// TIA Portal V18 export
// export: Created 2026-06-08T13:24:30.7103891Z, ExportSetting WithDefaults, DisplayName Totally Integrated Automation Portal, DisplayVersion V18, DisplayName TIA Portal Openness, DisplayVersion V18, DisplayName TIA Portal Version Control Interface, DisplayVersion V18, DisplayName STEP 7 Professional, DisplayVersion V18, DisplayName STEP 7 Safety, DisplayVersion V18, DisplayName WinCC Professional, DisplayVersion V18
ORGANIZATION_BLOCK "Main"   // OB1, LAD, ProgramCycle
TITLE = "Main Program Sweep (Cycle)"
{ S7_Optimized_Access := 'TRUE' }
VERSION : 0.1
// stored: AutoNumber true, IsIECCheckEnabled false, SetENOAutomatically false
   VAR_INPUT
      Initial_Call : Bool;   // Initial call of this OB
      Remanence : Bool;   // =True, if remanent data are available
   END_VAR
BEGIN

REGION Network 1: Modbus TCP Server - Call MB_SERVER
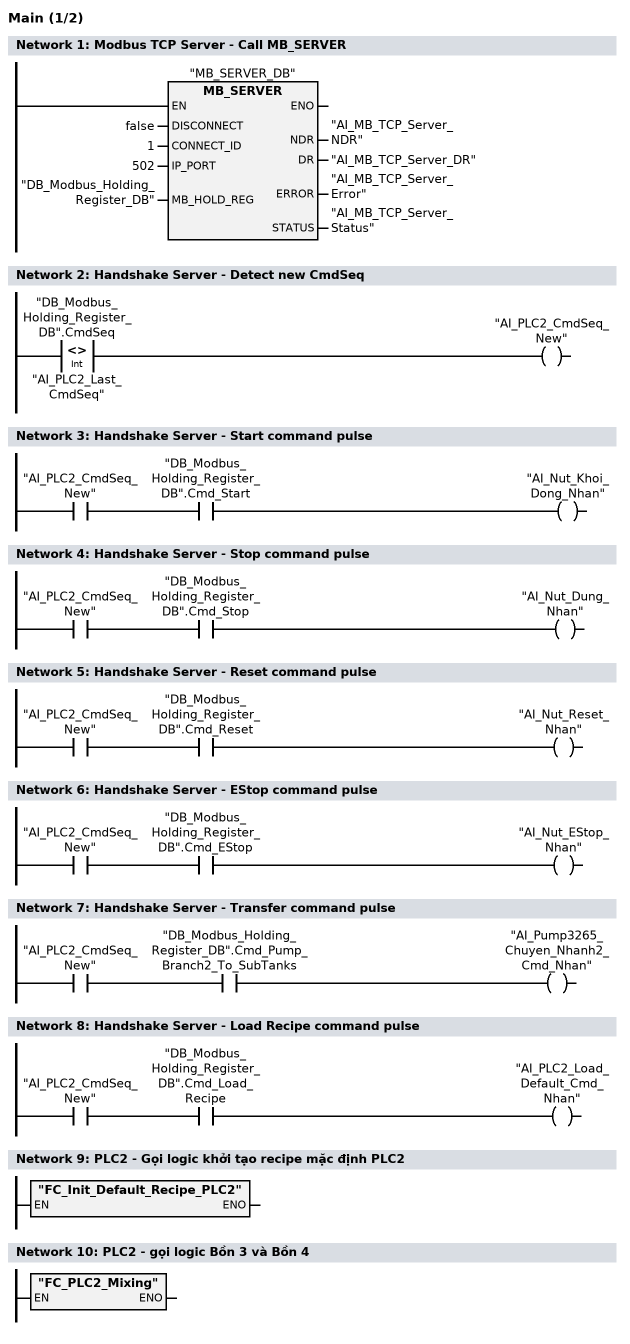
   RUNG wire#powerrail
      { S7_Templates := "[card1200 := 1, card1500 := 0]" } "MB_SERVER_DB".MB_SERVER(DISCONNECT := false, CONNECT_ID := 1, IP_PORT := 502, MB_HOLD_REG := "DB_Modbus_Holding_Register_DB", NDR => "AI_MB_TCP_Server_NDR", DR => "AI_MB_TCP_Server_DR", ERROR => "AI_MB_TCP_Server_Error", STATUS => "AI_MB_TCP_Server_Status")
   END_RUNG
   // the same network as SCL:
   "MB_SERVER_DB"(DISCONNECT := false,   // MB_SERVER
                  CONNECT_ID := 1,
                  IP_PORT := 502,
                  MB_HOLD_REG := "DB_Modbus_Holding_Register_DB",
                  NDR => "AI_MB_TCP_Server_NDR",
                  DR => "AI_MB_TCP_Server_DR",
                  ERROR => "AI_MB_TCP_Server_Error",
                  STATUS => "AI_MB_TCP_Server_Status");
END_REGION

REGION Network 2: Handshake Server - Detect new CmdSeq
   RUNG wire#powerrail
      { S7_Templates := "SrcType := Int" } NE_Contact(in1 := "DB_Modbus_Holding_Register_DB".CmdSeq, in2 := "AI_PLC2_Last_CmdSeq")
      Coil( "AI_PLC2_CmdSeq_New" )
   END_RUNG
   // the same network as SCL:
   "AI_PLC2_CmdSeq_New" := "DB_Modbus_Holding_Register_DB".CmdSeq <> "AI_PLC2_Last_CmdSeq";
END_REGION

REGION Network 3: Handshake Server - Start command pulse
   RUNG wire#powerrail
      Contact( "AI_PLC2_CmdSeq_New" )
      Contact( "DB_Modbus_Holding_Register_DB".Cmd_Start )
      Coil( "AI_Nut_Khoi_Dong_Nhan" )
   END_RUNG
   // the same network as SCL:
   "AI_Nut_Khoi_Dong_Nhan" := "AI_PLC2_CmdSeq_New" AND "DB_Modbus_Holding_Register_DB".Cmd_Start;
END_REGION

REGION Network 4: Handshake Server - Stop command pulse
   RUNG wire#powerrail
      Contact( "AI_PLC2_CmdSeq_New" )
      Contact( "DB_Modbus_Holding_Register_DB".Cmd_Stop )
      Coil( "AI_Nut_Dung_Nhan" )
   END_RUNG
   // the same network as SCL:
   "AI_Nut_Dung_Nhan" := "AI_PLC2_CmdSeq_New" AND "DB_Modbus_Holding_Register_DB".Cmd_Stop;
END_REGION

REGION Network 5: Handshake Server - Reset command pulse
   RUNG wire#powerrail
      Contact( "AI_PLC2_CmdSeq_New" )
      Contact( "DB_Modbus_Holding_Register_DB".Cmd_Reset )
      Coil( "AI_Nut_Reset_Nhan" )
   END_RUNG
   // the same network as SCL:
   "AI_Nut_Reset_Nhan" := "AI_PLC2_CmdSeq_New" AND "DB_Modbus_Holding_Register_DB".Cmd_Reset;
END_REGION

REGION Network 6: Handshake Server - EStop command pulse
   RUNG wire#powerrail
      Contact( "AI_PLC2_CmdSeq_New" )
      Contact( "DB_Modbus_Holding_Register_DB".Cmd_EStop )
      Coil( "AI_Nut_EStop_Nhan" )
   END_RUNG
   // the same network as SCL:
   "AI_Nut_EStop_Nhan" := "AI_PLC2_CmdSeq_New" AND "DB_Modbus_Holding_Register_DB".Cmd_EStop;
END_REGION

REGION Network 7: Handshake Server - Transfer command pulse
   RUNG wire#powerrail
      Contact( "AI_PLC2_CmdSeq_New" )
      Contact( "DB_Modbus_Holding_Register_DB".Cmd_Pump_Branch2_To_SubTanks )
      Coil( "AI_Pump3265_Chuyen_Nhanh2_Cmd_Nhan" )
   END_RUNG
   // the same network as SCL:
   "AI_Pump3265_Chuyen_Nhanh2_Cmd_Nhan" := "AI_PLC2_CmdSeq_New" AND "DB_Modbus_Holding_Register_DB".Cmd_Pump_Branch2_To_SubTanks;
END_REGION

REGION Network 8: Handshake Server - Load Recipe command pulse
   RUNG wire#powerrail
      Contact( "AI_PLC2_CmdSeq_New" )
      Contact( "DB_Modbus_Holding_Register_DB".Cmd_Load_Recipe )
      Coil( "AI_PLC2_Load_Default_Cmd_Nhan" )
   END_RUNG
   // the same network as SCL:
   "AI_PLC2_Load_Default_Cmd_Nhan" := "AI_PLC2_CmdSeq_New" AND "DB_Modbus_Holding_Register_DB".Cmd_Load_Recipe;
END_REGION

REGION Network 9: PLC2 - Gọi logic khởi tạo recipe mặc định PLC2
   RUNG wire#powerrail
      "FC_Init_Default_Recipe_PLC2"()
   END_RUNG
   // the same network as SCL:
   "FC_Init_Default_Recipe_PLC2"();
END_REGION

REGION Network 10: PLC2 - gọi logic Bồn 3 và Bồn 4
   RUNG wire#powerrail
      "FC_PLC2_Mixing"()
   END_RUNG
   // the same network as SCL:
   "FC_PLC2_Mixing"();
END_REGION

REGION Network 11: PLC2 - cập nhật mirror HMI
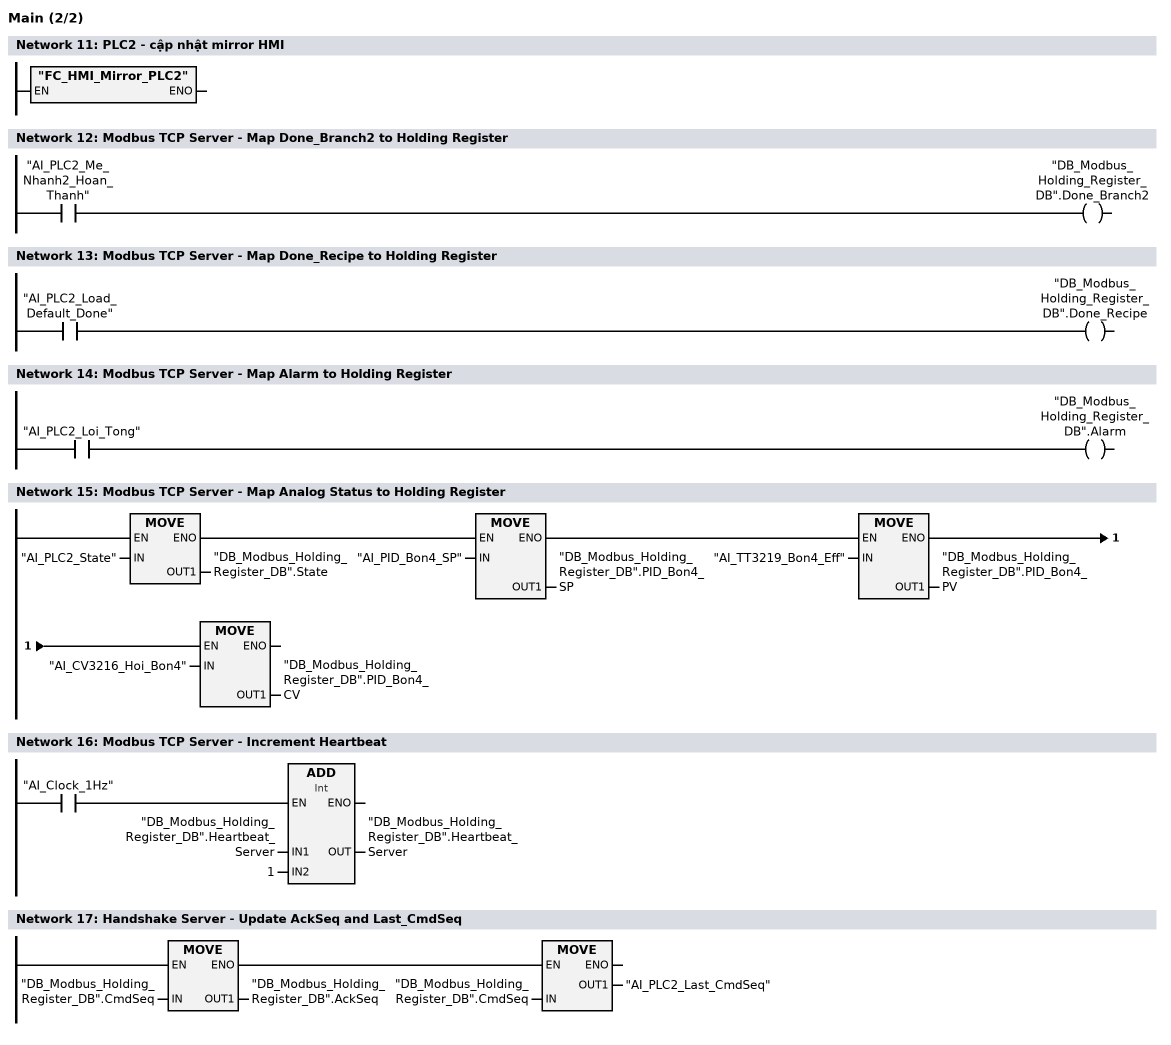
   RUNG wire#powerrail
      "FC_HMI_Mirror_PLC2"()
   END_RUNG
   // the same network as SCL:
   "FC_HMI_Mirror_PLC2"();
END_REGION

REGION Network 12: Modbus TCP Server - Map Done_Branch2 to Holding Register
   RUNG wire#powerrail
      Contact( "AI_PLC2_Me_Nhanh2_Hoan_Thanh" )
      Coil( "DB_Modbus_Holding_Register_DB".Done_Branch2 )
   END_RUNG
   // the same network as SCL:
   "DB_Modbus_Holding_Register_DB".Done_Branch2 := "AI_PLC2_Me_Nhanh2_Hoan_Thanh";
END_REGION

REGION Network 13: Modbus TCP Server - Map Done_Recipe to Holding Register
   RUNG wire#powerrail
      Contact( "AI_PLC2_Load_Default_Done" )
      Coil( "DB_Modbus_Holding_Register_DB".Done_Recipe )
   END_RUNG
   // the same network as SCL:
   "DB_Modbus_Holding_Register_DB".Done_Recipe := "AI_PLC2_Load_Default_Done";
END_REGION

REGION Network 14: Modbus TCP Server - Map Alarm to Holding Register
   RUNG wire#powerrail
      Contact( "AI_PLC2_Loi_Tong" )
      Coil( "DB_Modbus_Holding_Register_DB".Alarm )
   END_RUNG
   // the same network as SCL:
   "DB_Modbus_Holding_Register_DB".Alarm := "AI_PLC2_Loi_Tong";
END_REGION

REGION Network 15: Modbus TCP Server - Map Analog Status to Holding Register
   RUNG wire#powerrail
      { S7_GenerateENO := "TRUE" } Move(in := "AI_PLC2_State", out1 => "DB_Modbus_Holding_Register_DB".State)
      { S7_GenerateENO := "TRUE" } Move(in := "AI_PID_Bon4_SP", out1 => "DB_Modbus_Holding_Register_DB".PID_Bon4_SP)
      { S7_GenerateENO := "TRUE" } Move(in := "AI_TT3219_Bon4_Eff", out1 => "DB_Modbus_Holding_Register_DB".PID_Bon4_PV)
      { S7_GenerateENO := "TRUE" } Move(in := "AI_CV3216_Hoi_Bon4", out1 => "DB_Modbus_Holding_Register_DB".PID_Bon4_CV)
   END_RUNG
   // the same network as SCL:
   // ENO of a box is taken as its EN; it also drops when the box reports an error
   "DB_Modbus_Holding_Register_DB".State := "AI_PLC2_State";
   "DB_Modbus_Holding_Register_DB".PID_Bon4_SP := "AI_PID_Bon4_SP";
   "DB_Modbus_Holding_Register_DB".PID_Bon4_PV := "AI_TT3219_Bon4_Eff";
   "DB_Modbus_Holding_Register_DB".PID_Bon4_CV := "AI_CV3216_Hoi_Bon4";
END_REGION

REGION Network 16: Modbus TCP Server - Increment Heartbeat
   RUNG wire#powerrail
      Contact( "AI_Clock_1Hz" )
      { S7_Templates := "SrcType := Int"; S7_GenerateENO := "TRUE" } Add(in1 := "DB_Modbus_Holding_Register_DB".Heartbeat_Server, in2 := 1, out => "DB_Modbus_Holding_Register_DB".Heartbeat_Server)
   END_RUNG
   // the same network as SCL:
   IF "AI_Clock_1Hz" THEN
       "DB_Modbus_Holding_Register_DB".Heartbeat_Server := "DB_Modbus_Holding_Register_DB".Heartbeat_Server + 1;
   END_IF;
END_REGION

REGION Network 17: Handshake Server - Update AckSeq and Last_CmdSeq
   RUNG wire#powerrail
      { S7_GenerateENO := "TRUE" } Move(in := "DB_Modbus_Holding_Register_DB".CmdSeq, out1 => "DB_Modbus_Holding_Register_DB".AckSeq)
      { S7_GenerateENO := "TRUE" } Move(in := "DB_Modbus_Holding_Register_DB".CmdSeq, out1 => "AI_PLC2_Last_CmdSeq")
   END_RUNG
   // the same network as SCL:
   // ENO of a box is taken as its EN; it also drops when the box reports an error
   "DB_Modbus_Holding_Register_DB".AckSeq := "DB_Modbus_Holding_Register_DB".CmdSeq;
   "AI_PLC2_Last_CmdSeq" := "DB_Modbus_Holding_Register_DB".CmdSeq;
END_REGION
END_ORGANIZATION_BLOCK
